TYPE "udt_AccRollConveyor_COut_Manager"
VERSION : 0.1
// Block: udt_AccRollConveyor_COut_Manager
   STRUCT
      RollformerFeedOk : Bool;
      RollformerReqSlowDown : Bool;
      Empty : Bool;
      StopCut : Bool;
   END_STRUCT;

END_TYPE
